(* PLC project 05_timer.project, CODESYS CODESYS V3.5 SP22 Patch 2 *)
(* stored: creationDateTime 2026-07-23T20:51:32.9964433, modificationDateTime 2026-07-23T20:51:15.4134038 *)

PROGRAM PLC_PRG
  VAR
    fbTimer : TON;
    xEnable : BOOL;
    xDone : BOOL;
    tPreset : TIME := TIME#5s0ms;
    tElapsed : TIME;
    xTimerExecuted : BOOL;
  END_VAR

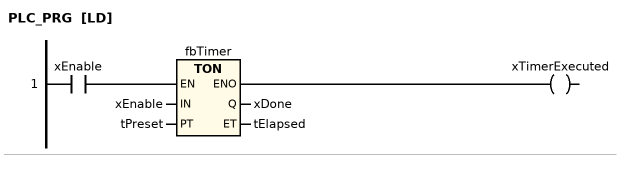
(* LD diagram, written out as Structured Text *)

fbTimer(EN := xEnable, IN := xEnable, PT := tPreset, Q => xDone, ET => tElapsed);
xTimerExecuted := fbTimer.ENO;
END_PROGRAM

CONFIGURATION Application
  RESOURCE Application ON PLC
    TASK MainTask(INTERVAL := T#20ms, PRIORITY := 1);
    PROGRAM PLC_PRG WITH MainTask : PLC_PRG;
  END_RESOURCE
END_CONFIGURATION
